// TIA Portal V19 export
DATA_BLOCK "Block_1_DB"   // DB4
// stored: InstanceOfName Block_1, InstanceOfType FB
"Block_1"
   // VAR_INPUT
   //    V1 : Bool;
   // END_VAR
   // VAR
   //    Program_Alarm_1 { S7_SetPoint := 'True'} : Program_Alarm;
   // END_VAR
BEGIN
END_DATA_BLOCK
